PROGRAM RunGrindingWheel
VAR
END_VAR

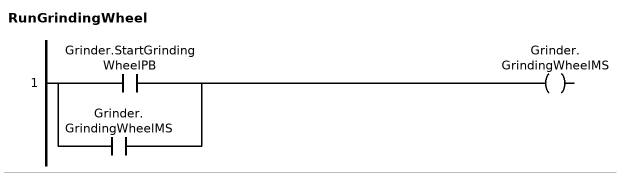
// NETWORK 1
Grinder.GrindingWheelMS := Grinder.StartGrindingWheelPB OR Grinder.GrindingWheelMS;

END_PROGRAM

(* stored: Version 1.1.0.1, ProductVersion 3.1.4024.4
   POU RunGrindingWheel: Id {3db83988-ca1e-4c38-a139-fd39660dbc4b}, SpecialFunc None *)
